PROGRAM Tests
VAR
    list_Person_Test : List_Person_Test;
    list_I_Observer_Test : List_I_Observer_Test;
END_VAR

TcUnit.RUN();

END_PROGRAM

(* stored: Version 1.1.0.1, ProductVersion 3.1.4024.6
   POU Tests: Id {27552b28-ca6c-444c-9236-5c59da3f3bc4}, SpecialFunc None *)
